TYPE ST_MovisafeCSBx1a_Config :
STRUCT	
	bSwapProcessData		: BOOL; //SWAP Process Data from/to FIELDBUS
END_STRUCT
END_TYPE

(* stored: Version 1.1.0.1, ProductVersion 3.1.4024.12
   DUT ST_MovisafeCSBx1a_Config: Id {8cc60221-2c88-09ff-0273-e729fcb5aebd} *)
